INTERFACE I_Halt EXTENDS I_StatusEx

PROPERTY CommandHalt : BOOL
SET
END_SET
END_PROPERTY

METHOD Halt
VAR_INPUT
    Deceleration : LREAL := 0.0;
    Jerk : LREAL := 0.0;
    BufferMode	: MC_BufferMode := MC_BufferMode.MC_Aborting;
END_VAR
END_METHOD

METHOD HaltDone
VAR_INPUT
END_VAR
END_METHOD

END_INTERFACE

(* stored: Version 1.1.0.1
   Itf I_Halt: Id {14029942-f501-4700-ae44-ffd198ee0804}
   Property CommandHalt: Id {5c8521dd-762c-4d7a-b33c-999816b31f14}
   Set Set: Id {323aeaa4-e9fd-40f3-904c-33931674b910}
   Method Halt: Id {d4ac7148-c266-4f03-80ec-1cc697d63c31}
   Method HaltDone: Id {98a490a7-8d10-42e3-b6a1-4ac74511a547} *)
